(* IEC 61131-3 sources: plcassist-cli/packages/volt-lsp-iec/test-corpus/bakon-nano/Device/Plc Logic/Application/POUs/Calculations/DataStorage, 3 files *)

(* ---- Stack_Init_CuttingPos.fun ---- *)
FUNCTION Stack_Init_CuttingPos : BOOL
VAR_INPUT
END_VAR
VAR_IN_OUT
	IQ_dataArray 		: ARRAY [*] OF XYA_Target;		//This has to be a reference to the actual array. (Underwater this is actually a pointer with dereferencing done for us.)
	IQ_dataArrayInfo	: ArrayInfo;
END_VAR
VAR
END_VAR

IQ_dataArrayInfo.index		:= DINT_TO_INT(LOWER_BOUND(IQ_dataArray, 1));
IQ_dataArrayInfo.lowerBound	:= DINT_TO_INT(LOWER_BOUND(IQ_dataArray, 1));
IQ_dataArrayInfo.upperbound	:= DINT_TO_INT(UPPER_BOUND(IQ_dataArray, 1));

Stack_Init_CuttingPos:= TRUE;
RETURN;

END_FUNCTION

(* ---- Stack_Push_CuttingPos.fun ---- *)
FUNCTION Stack_Push_CuttingPos : BOOL
//A stack functiones as a FILO buffer. The Push function pushes one item on the stack. (Pop is the counterpart.)
VAR_INPUT
	I_dataArray 		: POINTER TO XYA_Target;		//This has to be a pointer to the actual array.
END_VAR
VAR_IN_OUT
	IQ_dataArrayInfo	: ArrayInfo;
	IQ_item				: XYA_Target;
END_VAR
VAR

END_VAR

IF(IQ_dataArrayInfo.index < IQ_dataArrayInfo.lowerBound OR IQ_dataArrayInfo.index > IQ_dataArrayInfo.upperbound) THEN
	//The array is full.
	g_sMACH.ERR.bStackIsFull	:= TRUE;
	Stack_Push_CuttingPos := FALSE;
	RETURN;
END_IF

I_dataArray[IQ_dataArrayInfo.index - IQ_dataArrayInfo.lowerBound] := IQ_item;
IQ_dataArrayInfo.index := IQ_dataArrayInfo.index + 1;
Stack_Push_CuttingPos := TRUE;
RETURN;

END_FUNCTION

(* ---- StorePos.fun ---- *)
//Stores a cutting position to eather the cutting or waste table depending on the waste input bit.
FUNCTION StorePos : BOOL 						//Returns wether the position was sucessfully stored.

VAR CONSTANT
	defaultXYA 					: XYA_Target;	//A constant default XYA target
END_VAR
VAR_INPUT
	I_rX 						: REAL;			// X-pos
    I_rY 						: REAL;			// Y-pos
    I_rA 						: REAL;			// Rotation
    I_rK 						: REAL;			//
	I_bIsWaste					: BOOL;
	I_sOvershootSettings		: Gonio_Settings;
END_VAR
VAR
	sTempPosition		: XYA_Target;
END_VAR

sTempPosition 			:= defaultXYA;
sTempPosition.X_Target 	:= I_rX;
sTempPosition.Y_Target 	:= I_rY;
sTempPosition.A_Target 	:= I_rA;
sTempPosition.K_Target 	:= I_rK;

IF NOT Gonio_CorrectOvershoot(xya:=sTempPosition, settings:= I_sOvershootSettings) THEN
	g_sMACH.ERR.bOvershootCorrectionImpossible := TRUE;
	StorePos := g_HMI_MCH_Parameters.bSkipImpossiblePositions AND NOT g_sMACH.ERR.bMarginsInOvershootCorrectionInvalid AND NOT g_sMACH.ERR.bKnifeSettingsIncorrect AND NOT g_sMACH.ERR.bIntersectionNotFound;
	RETURN;
END_IF

StorePos := SEL(I_bIsWaste,	Stack_Push_CuttingPos(I_dataArray := ADR(g_aCuttingPositions), 	IQ_dataArrayInfo := g_sCuttingPositionsInfo,	IQ_item := sTempPosition),
							Stack_Push_CuttingPos(I_dataArray := ADR(g_aWastePositions), 	IQ_dataArrayInfo := g_sWastePositionsInfo, 		IQ_item := sTempPosition));

RETURN;

END_FUNCTION
